FUNCTION_BLOCK FB_Valve53_Ctrl
VAR_INPUT
	i_bInterlock		:BOOL;
	i_bProcesslock		:BOOL;
	i_bCmd_Disable		:BOOL;
	i_bCmd_Close		:BOOL;
	i_bCmd_HalfOpen		:BOOL;
	i_bCmd_Open			:BOOL;
	i_bSensorClosed		:BOOL;
	i_bSensorHalfOpen	:BOOL;
	i_bSensorOpen		:BOOL;
	i_tTimeout			:TIME;
	i_tTimeOutHalf		:TIME;
END_VAR
VAR_OUTPUT
	q_bCmd_Release		:BOOL;
	q_bCmd_Close		:BOOL;
	q_bCmd_Open			:BOOL;
	q_bEnabled			:BOOL;
	q_bClosed			:BOOL;
	q_bHalfOpened		:BOOL;
	q_bOpened			:BOOL;
	q_bTraveling		:BOOL;
	q_bClose_Timeout	:BOOL;
	q_bOpen_Timeout		:BOOL;
	q_bHOpen_Timeout	:BOOL;
END_VAR
VAR
	tonTimeoutClose		:TON;
	tonTimeOutHOpen		:TON;
	tonTimeoutOpen		:TON;
	bMidPosReq			:BOOL;
END_VAR
VAR // added by the converter: edge detectors and wires of the graphical bodies
    _rt1, _rt2, _rt3 : R_TRIG;
    _w1, _w2, _w3, _w4, _w5 : BOOL;
END_VAR

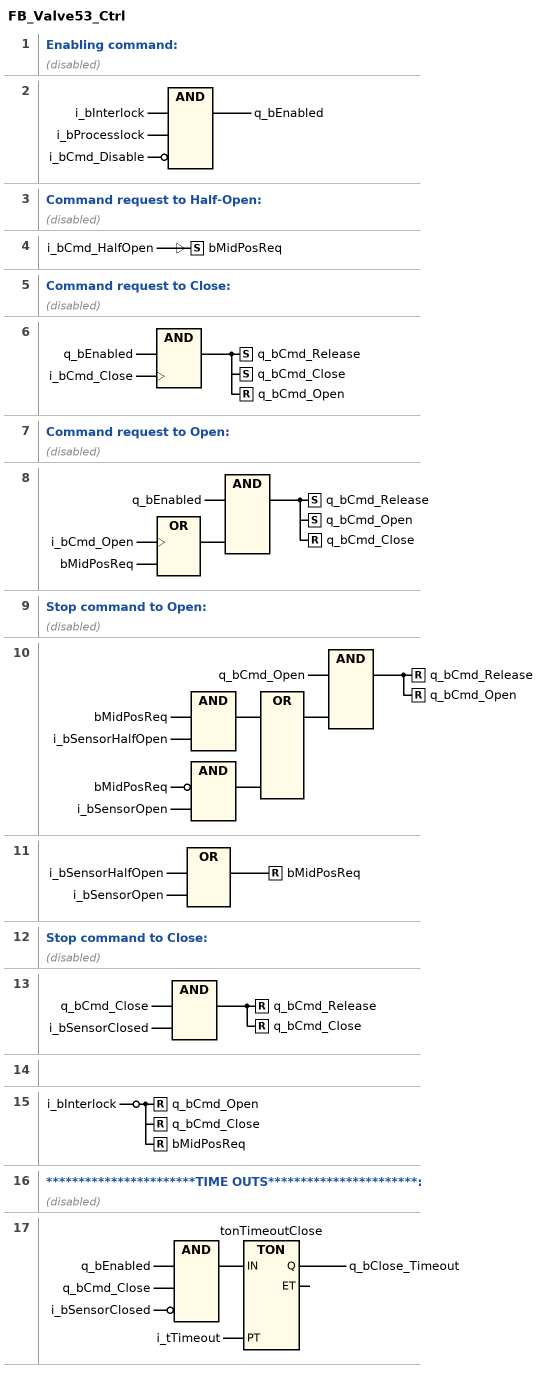
// NETWORK 1 (disabled)
// label: Enabling command

// NETWORK 2
q_bEnabled := i_bInterlock AND i_bProcesslock AND NOT i_bCmd_Disable;

// NETWORK 3 (disabled)
// label: Command request to Half-Open

// NETWORK 4
_rt1(CLK := i_bCmd_HalfOpen);
bMidPosReq S= _rt1.Q;

// NETWORK 5 (disabled)
// label: Command request to Close

// NETWORK 6
_rt2(CLK := i_bCmd_Close);
_w1 := q_bEnabled AND _rt2.Q;
q_bCmd_Release S= _w1;
q_bCmd_Close S= _w1;
q_bCmd_Open R= _w1;

// NETWORK 7 (disabled)
// label: Command request to Open

// NETWORK 8
_rt3(CLK := i_bCmd_Open);
_w2 := q_bEnabled AND (_rt3.Q OR bMidPosReq);
q_bCmd_Release S= _w2;
q_bCmd_Open S= _w2;
q_bCmd_Close R= _w2;

// NETWORK 9 (disabled)
// label: Stop command to Open

// NETWORK 10
_w3 := q_bCmd_Open AND (bMidPosReq AND i_bSensorHalfOpen OR NOT bMidPosReq AND i_bSensorOpen);
q_bCmd_Release R= _w3;
q_bCmd_Open R= _w3;

// NETWORK 11
bMidPosReq R= i_bSensorHalfOpen OR i_bSensorOpen;

// NETWORK 12 (disabled)
// label: Stop command to Close

// NETWORK 13
_w4 := q_bCmd_Close AND i_bSensorClosed;
q_bCmd_Release R= _w4;
q_bCmd_Close R= _w4;

// NETWORK 14

// NETWORK 15
_w5 := NOT i_bInterlock;
q_bCmd_Open R= _w5;
q_bCmd_Close R= _w5;
bMidPosReq R= _w5;

// NETWORK 16 (disabled)
// label: ***********************TIME OUTS***********************

// NETWORK 17
tonTimeoutClose(IN := q_bEnabled AND q_bCmd_Close AND NOT i_bSensorClosed, PT := i_tTimeout); // TON
q_bClose_Timeout := tonTimeoutClose.Q;

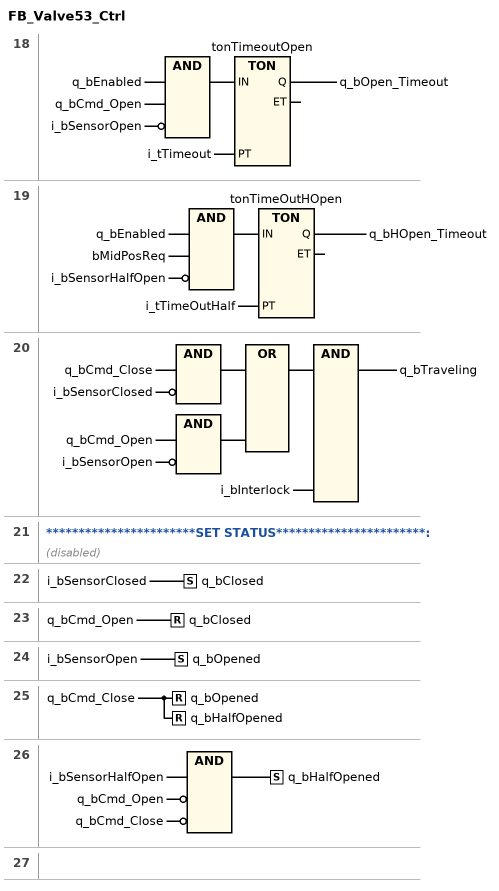
// NETWORK 18
tonTimeoutOpen(IN := q_bEnabled AND q_bCmd_Open AND NOT i_bSensorOpen, PT := i_tTimeout); // TON
q_bOpen_Timeout := tonTimeoutOpen.Q;

// NETWORK 19
tonTimeOutHOpen(IN := q_bEnabled AND bMidPosReq AND NOT i_bSensorHalfOpen, PT := i_tTimeOutHalf); // TON
q_bHOpen_Timeout := tonTimeOutHOpen.Q;

// NETWORK 20
q_bTraveling := (q_bCmd_Close AND NOT i_bSensorClosed OR q_bCmd_Open AND NOT i_bSensorOpen) AND i_bInterlock;

// NETWORK 21 (disabled)
// label: ***********************SET STATUS***********************

// NETWORK 22
q_bClosed S= i_bSensorClosed;

// NETWORK 23
q_bClosed R= q_bCmd_Open;

// NETWORK 24
q_bOpened S= i_bSensorOpen;

// NETWORK 25
q_bOpened R= q_bCmd_Close;
q_bHalfOpened R= q_bCmd_Close;

// NETWORK 26
q_bHalfOpened S= i_bSensorHalfOpen AND NOT q_bCmd_Open AND NOT q_bCmd_Close;

// NETWORK 27

END_FUNCTION_BLOCK

(* stored: Version 1.1.0.1, ProductVersion 3.1.4024.12
   POU FB_Valve53_Ctrl: Id {53314072-cfa1-44e5-9fa5-54acb762f89b}, SpecialFunc None *)
